Fanuc KAREL source: kt00224.KL

PROGRAM KT00224
%STACKSIZE=65535
%PRIORITY=65535
%NOLOCKGROUP
VAR
H1 : ARRAY[2] OF SHORT
H2 : ARRAY[2] OF SHORT
OUT : INTEGER
BEGIN
H1[1]=2
H2[1]=3
H1[1]=2
H2[1]=3
-- UNRESOLVED_PC line 12 opcodes [22 9D 33 B3 22 9D 33 B3 46 23] marker_code=76
END KT00224
